FUNCTION_BLOCK FB_PressSectionDriveControl_V2_bak

VAR_INPUT

    //────────────────────────────────────────────
    // GROUP / INTERLOCKS
    //────────────────────────────────────────────
    startGroup              : BOOL; // Start command (pulse) / Comando de partida (pulso)
    stopGroup               : BOOL; // Stop command (level) / Comando de parada (nível)
    groupReset              : BOOL; // Fault reset / Reset de falhas do grupo
	
    //────────────────────────────────────────────
    // AUXILIARY MOTORS — INDICATORS & COMMANDS
    //────────────────────────────────────────────
    grouSpeedDifIncCmd         : BOOL; // Lamp: offset increasing / Lâmpada: aumento de offset
    grouSpeedDifDecCmd         : BOOL; // Lamp: offset decreasing / Lâmpada: redução de offset
	
    //────────────────────────────────────────────
    // SPEED ADJUSTMENTS / OFFSET TUNING
    //────────────────────────────────────────────
    groupRecoverSpeedCmd    : BOOL; // Recover speed while TRUE / Recuperar velocidade enquanto TRUE


    //────────────────────────────────────────────
    // DRIVE STATUS INPUTS — PRESS SECTION (2 MOTORS)
    //────────────────────────────────────────────
    firstPressReady         : BOOL; // First press (MASTER) ready / Prensa 1 (mestre) pronto
    secondPressReady        : BOOL; // Second press (SLAVE) ready / Prensa 2 (escravo) pronto

    //────────────────────────────────────────────
    // SPEED SETPOINTS / MODE
    //────────────────────────────────────────────
    groupAutoSpeedMPM       : REAL; // Auto mode speed [m/min] / Velocidade em modo automático [m/min]
    groupManualSpeedMPM     : REAL := 50.0; // Manual mode speed / Velocidade em modo manual
    groupSpeedAutoMan       : BOOL; // Speed mode: 0=Manual, 1=Auto / Modo de velocidade: 0=Manual, 1=Automático

    //────────────────────────────────────────────
    // SPEED & TORQUE FEEDBACKS
    //────────────────────────────────────────────
    firstPressSpeedFeedback : REAL; // First press speed feedback / Velocidade medida da prensa 1
    firstPressTorqueFeedback: REAL; // First press torque feedback / Torque da prensa 1
    secondPressSpeedFeedback: REAL; // Second press speed feedback / Velocidade medida da prensa 2
    secondPressTorqueFeedback: REAL; // Second press torque feedback / Torque da prensa 2


    //──── Upper Felt 1 Stretcher ────
    upperFelt1StretcherCmdFwd     : BOOL; // Run forward / Comando para frente
    upperFelt1StretcherCmdRev     : BOOL; // Run reverse / Comando para trás
    upperFelt1StretcherFault      : BOOL; // Fault detected / Falha detectada
    upperFelt1StretcherLimitFwd   : BOOL; // End limit forward / Fim de curso frente
    upperFelt1StretcherLimitRev   : BOOL; // End limit reverse / Fim de curso trás

    //──── Upper Felt 2 Stretcher ────
    upperFelt2StretcherCmdFwd     : BOOL; // Run forward / Comando para frente
    upperFeltt2tretcherCmdRev     : BOOL; // Run reverse / Comando para trás (corrigir nome!)
    upperFeltS2tretcherFault      : BOOL; // Fault detected / Falha detectada
    upperFeltS2tretcherLimitFwd   : BOOL; // End limit forward / Fim de curso frente
    upperFeltS2tretcherLimitRev   : BOOL; // End limit reverse / Fim de curso trás

    //──── Lower Felt Stretcher ────
    lowerFeltStretcherCmdFwd      : BOOL;
    lowerFeltStretcherCmdRev      : BOOL;
    lowerFeltStretcherFault       : BOOL;
    lowerFeltStretcherLimitFwd    : BOOL;
    lowerFeltStretcherLimitRev    : BOOL;

    //──── Upper Infeed Roll ────
    upperInfeedRollCmdFwd         : BOOL;
    upperInfeedRollCmdRev         : BOOL;
    upperInfeedRollFault          : BOOL;
    upperInfeedRollLimitFwd       : BOOL;
    upperInfeedRollLimitRev       : BOOL;

    //──── Lower Infeed Roll ────
    lowerInfeedRollCmdFwd         : BOOL;
    lowerInfeedRollCmdRev         : BOOL;
    lowerInfeedRollFault          : BOOL;
    lowerInfeedRollLimitFwd       : BOOL;
    lowerInfeedRollLimitRev       : BOOL;

    //────────────────────────────────────────────
    // FELT EDGE / RUNNING SAFETY SENSORS
    //────────────────────────────────────────────
    pressSectionUpperFelt1OverrunSensorOperatorSide : BOOL; // Operator side / Lado operador
    pressSectionUpperFelt1OverrunSensorDriveSide    : BOOL; // Drive side / Lado comando

    pressSectionUpperFelt2OverrunSensorOperatorSide : BOOL;
    pressSectionUpperFelt2OverrunSensorDriveSide    : BOOL;

    pressSectionLowerFeltOverrunSensorOperatorSide  : BOOL;
    pressSectionLowerFeltOverrunSensorDriveSide     : BOOL;

	
	machineConfig			:  PaperMachine_TypeHmiConfig;
	
END_VAR



VAR_OUTPUT

    //────────────────────────────────────────────
    // STATE / DIAGNOSTICS
    //────────────────────────────────────────────
    deviceState                 : STRING; // Current state string / Estado atual em texto
    statusCode                  : INT;    // 0=Idle, 1=Starting, 2=Running, 3=Fault
    groupFault                  : BOOL;   // TRUE if any group fault active / Falha geral do grupo


    //────────────────────────────────────────────
    // SPEED REFERENCES (TO DRIVES) AND DISPLAY
    //────────────────────────────────────────────
    firstPressSpeedSetpointRPM  		: REAL; // Master speed reference [%] / Referência de velocidade mestre
    secondPressSpeedSetpointRPM 		: REAL; // Slave speed reference [%] / Referência de velocidade escravo 
	
	firstPressSpeedFeedbackRPM  		: REAL; // Master speed reference [%] / Referência de velocidade mestre
    secondPressSpeedFeedbackRPM 		: REAL; // Slave speed reference [%] / Referência de velocidade escravo 
	
	firstPressSpeedFeedbackMPM  		: REAL; // Master speed reference [%] / Referência de velocidade mestre
    secondPressSpeedFeedbackMPM 		: REAL; // Slave speed reference [%] / Referência de velocidade escravo 

	firstPressTorqueFeedbackPct  		: REAL; // Master speed reference [%] / Referência de velocidade mestre
    secondPressTorqueFeedbackPct 		: REAL; // Slave speed reference [%] / Referência de velocidade escravo 
	
	
	nextGroupSpeedRefMPM        : REAL; // Next group speed [m/min] / Velocidade do próximo grupo [m/min]

    //────────────────────────────────────────────
    // TORQUE REFERENCES / LIMITS (SLAVE)
    //────────────────────────────────────────────
    firstPressTorqueRefPct : REAL; // Torque setpoint for slave / Referência de torque escravo

    //────────────────────────────────────────────
    // DRIVE COMMANDS (ENABLE / RESET)
    //────────────────────────────────────────────
    firstPressDriveEnable        : BOOL; // Enable master drive / Habilita drive mestre
    firstPressDriveReset         : BOOL; // Reset master drive fault / Reset falha drive mestre
    secondPressDriveEnable       : BOOL; // Enable slave drive / Habilita drive escravo
    secondPressDriveReset        : BOOL; // Reset slave drive fault / Reset falha drive escravo

    //────────────────────────────────────────────
    // STATUS CODES (PER DRIVE)
    //────────────────────────────────────────────
    firstPressStatusCode        : INT; // 0=Idle, 1=Start, 2=Run, 3=Fault / Código de status da prensa 1
    secondPressStatusCode       : INT; // Código de status da prensa 2

    //────────────────────────────────────────────
    // AUXILIARY MOTORS — DIRECT START OUTPUTS
    //────────────────────────────────────────────
    upperFelt1StretcherRunFwd   : BOOL; // Run forward / Rodar para frente
    upperFelt1StretcherRunRev   : BOOL; // Run reverse / Rodar para trás

    upperFelt2StretcherRunFwd   : BOOL;
    upperFelt2StretcherRunRev   : BOOL;

    lowerFeltStretcherRunFwd    : BOOL;
    lowerFeltStretcherRunRev    : BOOL;

    upperInfeedRollRunFwd       : BOOL;
    upperInfeedRollRunRev       : BOOL;

    lowerInfeedRollRunFwd       : BOOL;
    lowerInfeedRollRunRev       : BOOL;

    //────────────────────────────────────────────
    // HMI ALARMS STRUCTURE
    //────────────────────────────────────────────
    hmiAlarms                   : PaperMachine_TypeHmiAlarms; // Alarm structure / Estrutura de alarmes

END_VAR




VAR
 
	instFB_GroupDriveControl_V1 : FB_GroupDriveControl_V1;
	instFB_GroupSpeedControl_V1 : FB_GroupSpeedControl_V1;
	instFB_GroupDisplayFilters_V1 : FB_GroupDisplayFilters_V1;
	instFB_GroupTorqueTrimControl_V1 : FB_GroupTorqueTrimControl_V1;

	instFB_GroupTorqueTrimControl_V2: FB_GroupTorqueTrimControl_V2;
	speedDif: REAL;
	speedDifError: BOOL;
END_VAR

VAR PERSISTENT

END_VAR

// ─────────────────────────────────────────────────────────────────────────────
// MAIN CALL SEQUENCE
// ─────────────────────────────────────────────────────────────────────────────

_GroupControl();          // 1) State machine: edges, enables, stop modes
_StateDisplay();
_SpeedDifferenceCheck();  // 4) Speed difference monitor & trip
_auxiliaryControls();

_alarmsDisplay();

METHOD _alarmsDisplay
VAR_INPUT
END_VAR
(*
//==============================================================
// FAULT EVALUATION — PER CONDITION (flags only; no global set)
//==============================================================

//----------------------------
// PRESS SECTION DRIVES
//----------------------------
hmiAlarms.pressSectionFirstPressFaultAlarm  := firstPressVfdFaultFeedback;
hmiAlarms.pressSectionSecondPressFaultAlarm := secondPressVfdFaultFeedback;

//----------------------------
// PRESS SECTION AUXILIARIES
//----------------------------
hmiAlarms.pressSectionUpperFeltStretcherFaultAlarm := upperFelt1StretcherFault;
hmiAlarms.pressSectionLowerFeltStretcherFaultAlarm := lowerFeltStretcherFault;
hmiAlarms.pressSectionUpperInfeedRollFaultAlarm    := upperInfeedRollFault;
hmiAlarms.pressSectionLowerInfeedRollFaultAlarm    := lowerInfeedRollFault;


//==============================================================
// PRESS SECTION — FELT EDGE OVERRUN ALARMS (DIRECT SENSORS)
//==============================================================

hmiAlarms.pressSectionUpperFelt1OverrunOperatorSideAlarm := pressSectionUpperFelt1OverrunSensorOperatorSide;
hmiAlarms.pressSectionUpperFelt1OverrunDriveSideAlarm    := pressSectionUpperFelt1OverrunSensorDriveSide;

hmiAlarms.pressSectionUpperFelt2OverrunOperatorSideAlarm := pressSectionUpperFelt2OverrunSensorOperatorSide;
hmiAlarms.pressSectionUpperFelt2OverrunDriveSideAlarm    := pressSectionUpperFelt2OverrunSensorDriveSide;

hmiAlarms.pressSectionLowerFeltOverrunOperatorSideAlarm := pressSectionLowerFeltOverrunSensorOperatorSide;
hmiAlarms.pressSectionLowerFeltOverrunDriveSideAlarm    := pressSectionLowerFeltOverrunSensorDriveSide;


//----------------------------
// PRESS SECTION GROUP FAULT STATUS
//----------------------------
groupFault :=
    hmiAlarms.pressSectionFirstPressFaultAlarm 
	OR hmiAlarms.pressSectionSecondPressFaultAlarm 
	OR hmiAlarms.pressFelt1OverrunOperatorSideAlarm
	OR hmiAlarms.pressFelt1OverrunDriveSideAlarm
	OR hmiAlarms.pressFelt2OverrunOperatorSideAlarm
	OR hmiAlarms.pressFelt2OverrunDriveSideAlarm
	OR hmiAlarms.pressFelt3OverrunOperatorSideAlarm
	OR hmiAlarms.pressFelt3OverrunDriveSideAlarm;


*)
//==============================================================
// FAULT EVALUATION — PER CONDITION (flags only; no global set)
//==============================================================

//----------------------------
// PRESS SECTION DRIVES
//----------------------------
//hmiAlarms.pressSectionFirstPressFaultAlarm  := firstPressVfdFaultFeedback;
//hmiAlarms.pressSectionSecondPressFaultAlarm := secondPressVfdFaultFeedback;

//----------------------------
// PRESS SECTION AUXILIARIES
//----------------------------
hmiAlarms.pressSectionUpperFeltStretcherFaultAlarm := upperFelt1StretcherFault;
hmiAlarms.pressSectionLowerFeltStretcherFaultAlarm := lowerFeltStretcherFault;
hmiAlarms.pressSectionUpperInfeedRollFaultAlarm    := upperInfeedRollFault;
hmiAlarms.pressSectionLowerInfeedRollFaultAlarm    := lowerInfeedRollFault;


//==============================================================
// PRESS SECTION — FELT EDGE OVERRUN ALARMS (DIRECT SENSORS)
//==============================================================

hmiAlarms.pressSectionUpperFelt1OverrunOperatorSideAlarm := pressSectionUpperFelt1OverrunSensorOperatorSide;
hmiAlarms.pressSectionUpperFelt1OverrunDriveSideAlarm    := pressSectionUpperFelt1OverrunSensorDriveSide;

hmiAlarms.pressSectionUpperFelt2OverrunOperatorSideAlarm := pressSectionUpperFelt2OverrunSensorOperatorSide;
hmiAlarms.pressSectionUpperFelt2OverrunDriveSideAlarm    := pressSectionUpperFelt2OverrunSensorDriveSide;

hmiAlarms.pressSectionLowerFeltOverrunOperatorSideAlarm := pressSectionLowerFeltOverrunSensorOperatorSide;
hmiAlarms.pressSectionLowerFeltOverrunDriveSideAlarm    := pressSectionLowerFeltOverrunSensorDriveSide;


//----------------------------
// PRESS SECTION GROUP FAULT STATUS
//----------------------------
groupFault := hmiAlarms.pressSectionFirstPressFaultAlarm OR
		hmiAlarms.pressSectionSecondPressFaultAlarm OR
		hmiAlarms.pressSectionUpperFelt1OverrunOperatorSideAlarm OR
		hmiAlarms.pressSectionUpperFelt1OverrunDriveSideAlarm OR
		hmiAlarms.pressSectionUpperFelt2OverrunOperatorSideAlarm OR
		hmiAlarms.pressSectionUpperFelt2OverrunDriveSideAlarm OR
		hmiAlarms.pressSectionLowerFeltOverrunOperatorSideAlarm OR
		hmiAlarms.pressSectionLowerFeltOverrunDriveSideAlarm;
END_METHOD

METHOD _auxiliaryControls
VAR_INPUT
END_VAR
//============================
// LOWER FELT STRETCHER
//============================
IF NOT lowerFeltStretcherFault THEN
    IF lowerFeltStretcherCmdFwd AND NOT lowerFeltStretcherCmdRev AND NOT lowerFeltStretcherLimitFwd THEN
        lowerFeltStretcherRunFwd := TRUE;
    ELSE
        lowerFeltStretcherRunFwd := FALSE;
    END_IF;

    IF lowerFeltStretcherCmdRev AND NOT lowerFeltStretcherCmdFwd AND NOT lowerFeltStretcherLimitRev THEN
        lowerFeltStretcherRunRev := TRUE;
    ELSE
        lowerFeltStretcherRunRev := FALSE;
    END_IF;
ELSE
    lowerFeltStretcherRunFwd := FALSE;
    lowerFeltStretcherRunRev := FALSE;
END_IF;


//============================
// UPPER INFEED ROLL
//============================
IF NOT upperInfeedRollFault THEN
    IF upperInfeedRollCmdFwd AND NOT upperInfeedRollCmdRev AND NOT upperInfeedRollLimitFwd THEN
        upperInfeedRollRunFwd := TRUE;
    ELSE
        upperInfeedRollRunFwd := FALSE;
    END_IF;

    IF upperInfeedRollCmdRev AND NOT upperInfeedRollCmdFwd AND NOT upperInfeedRollLimitRev THEN
        upperInfeedRollRunRev := TRUE;
    ELSE
        upperInfeedRollRunRev := FALSE;
    END_IF;
ELSE
    upperInfeedRollRunFwd := FALSE;
    upperInfeedRollRunRev := FALSE;
END_IF;


//============================
// LOWER INFEED ROLL
//============================
IF NOT lowerInfeedRollFault THEN
    IF lowerInfeedRollCmdFwd AND NOT lowerInfeedRollCmdRev AND NOT lowerInfeedRollLimitFwd THEN
        lowerInfeedRollRunFwd := TRUE;
    ELSE
        lowerInfeedRollRunFwd := FALSE;
    END_IF;

    IF lowerInfeedRollCmdRev AND NOT lowerInfeedRollCmdFwd AND NOT lowerInfeedRollLimitRev THEN
        lowerInfeedRollRunRev := TRUE;
    ELSE
        lowerInfeedRollRunRev := FALSE;
    END_IF;
ELSE
    lowerInfeedRollRunFwd := FALSE;
    lowerInfeedRollRunRev := FALSE;
END_IF;


//============================
// UPPER FELT 1 STRETCHER
//============================
IF NOT upperFelt1StretcherFault THEN
    IF upperFelt1StretcherCmdFwd AND NOT upperFelt1StretcherCmdRev AND NOT upperFelt1StretcherLimitFwd THEN
        upperFelt1StretcherRunFwd := TRUE;
    ELSE
        upperFelt1StretcherRunFwd := FALSE;
    END_IF;

    IF upperFelt1StretcherCmdRev AND NOT upperFelt1StretcherCmdFwd AND NOT upperFelt1StretcherLimitRev THEN
        upperFelt1StretcherRunRev := TRUE;
    ELSE
        upperFelt1StretcherRunRev := FALSE;
    END_IF;
ELSE
    upperFelt1StretcherRunFwd := FALSE;
    upperFelt1StretcherRunRev := FALSE;
END_IF;

//============================
// UPPER FELT 2 STRETCHER
//============================
IF NOT upperFeltS2tretcherFault THEN
    IF upperFelt2StretcherCmdFwd AND NOT upperFeltt2tretcherCmdRev AND NOT upperFeltS2tretcherLimitFwd THEN
        upperFelt2StretcherRunFwd := TRUE;
    ELSE
        upperFelt2StretcherRunFwd := FALSE;
    END_IF;

    IF upperFeltt2tretcherCmdRev AND NOT upperFelt2StretcherCmdFwd AND NOT upperFeltS2tretcherLimitRev THEN
        upperFelt2StretcherRunRev := TRUE;
    ELSE
        upperFelt2StretcherRunRev := FALSE;
    END_IF;
ELSE
    upperFelt2StretcherRunFwd := FALSE;
    upperFelt2StretcherRunRev := FALSE;
END_IF;
END_METHOD

METHOD _GroupControl
VAR_INPUT
END_VAR
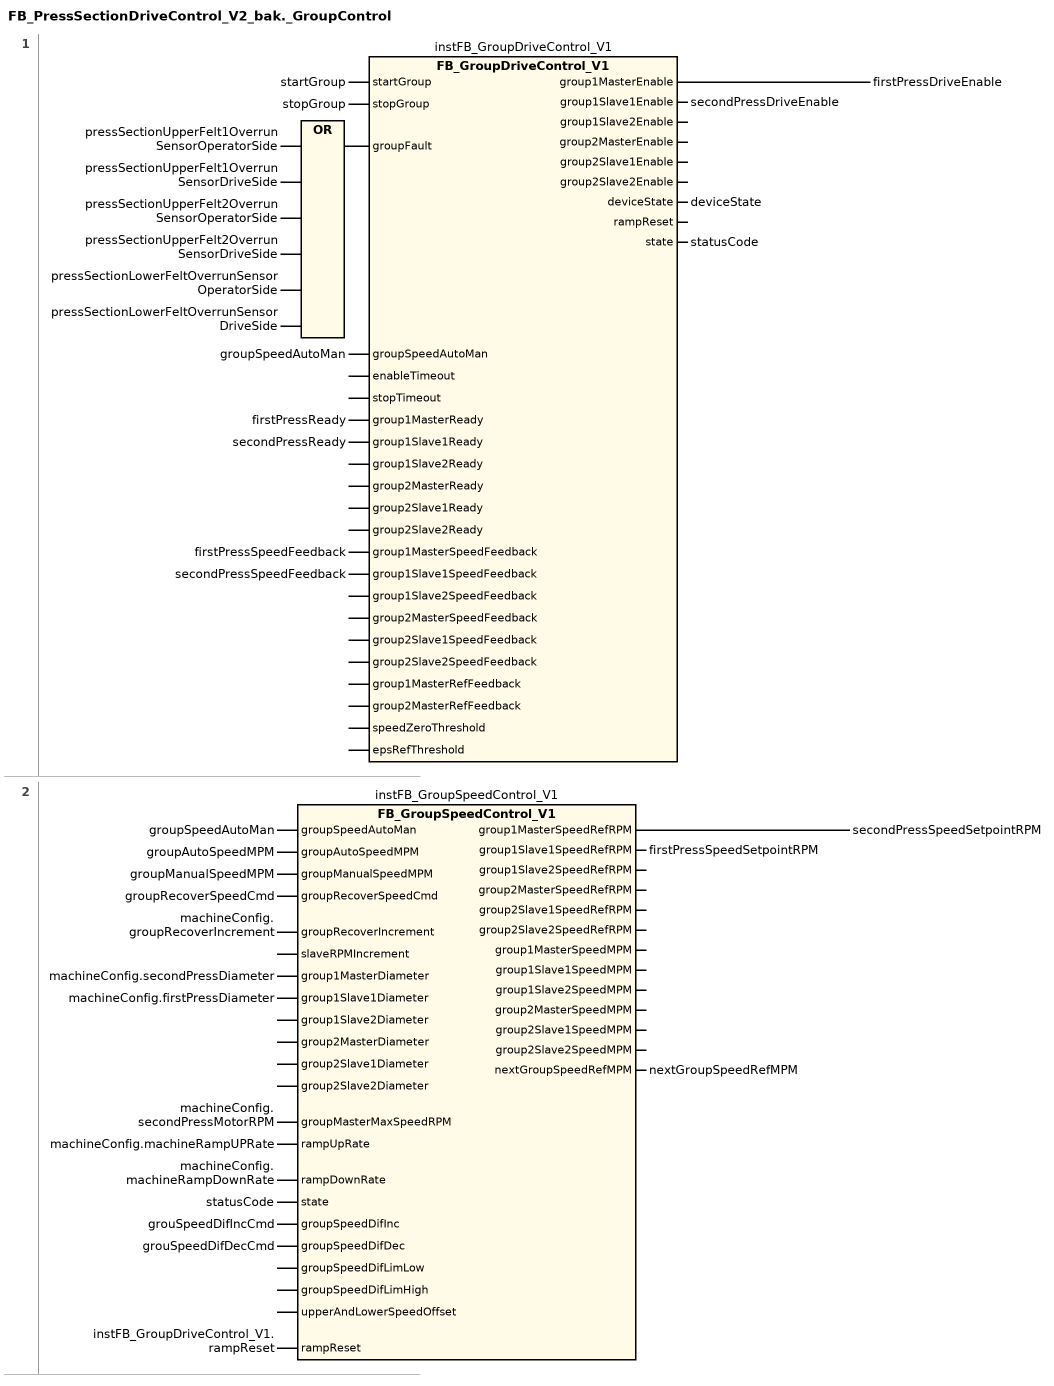
// NETWORK 1
instFB_GroupDriveControl_V1(
    startGroup := startGroup,
    stopGroup := stopGroup,
    groupFault := pressSectionUpperFelt1OverrunSensorOperatorSide OR pressSectionUpperFelt1OverrunSensorDriveSide OR pressSectionUpperFelt2OverrunSensorOperatorSide OR pressSectionUpperFelt2OverrunSensorDriveSide OR pressSectionLowerFeltOverrunSensorOperatorSide OR pressSectionLowerFeltOverrunSensorDriveSide,
    groupSpeedAutoMan := groupSpeedAutoMan,
    group1MasterReady := firstPressReady,
    group1Slave1Ready := secondPressReady,
    group1MasterSpeedFeedback := firstPressSpeedFeedback,
    group1Slave1SpeedFeedback := secondPressSpeedFeedback,
    group1Slave1Enable => secondPressDriveEnable,
    deviceState => deviceState,
    state => statusCode); // FB_GroupDriveControl_V1
firstPressDriveEnable := instFB_GroupDriveControl_V1.group1MasterEnable;

// NETWORK 2
instFB_GroupSpeedControl_V1(
    groupSpeedAutoMan := groupSpeedAutoMan,
    groupAutoSpeedMPM := groupAutoSpeedMPM,
    groupManualSpeedMPM := groupManualSpeedMPM,
    groupRecoverSpeedCmd := groupRecoverSpeedCmd,
    groupRecoverIncrement := machineConfig.groupRecoverIncrement,
    group1MasterDiameter := machineConfig.secondPressDiameter,
    group1Slave1Diameter := machineConfig.firstPressDiameter,
    groupMasterMaxSpeedRPM := machineConfig.secondPressMotorRPM,
    rampUpRate := machineConfig.machineRampUPRate,
    rampDownRate := machineConfig.machineRampDownRate,
    state := statusCode,
    groupSpeedDifInc := grouSpeedDifIncCmd,
    groupSpeedDifDec := grouSpeedDifDecCmd,
    rampReset := instFB_GroupDriveControl_V1.rampReset,
    group1Slave1SpeedRefRPM => firstPressSpeedSetpointRPM,
    nextGroupSpeedRefMPM => nextGroupSpeedRefMPM); // FB_GroupSpeedControl_V1
secondPressSpeedSetpointRPM := instFB_GroupSpeedControl_V1.group1MasterSpeedRefRPM;

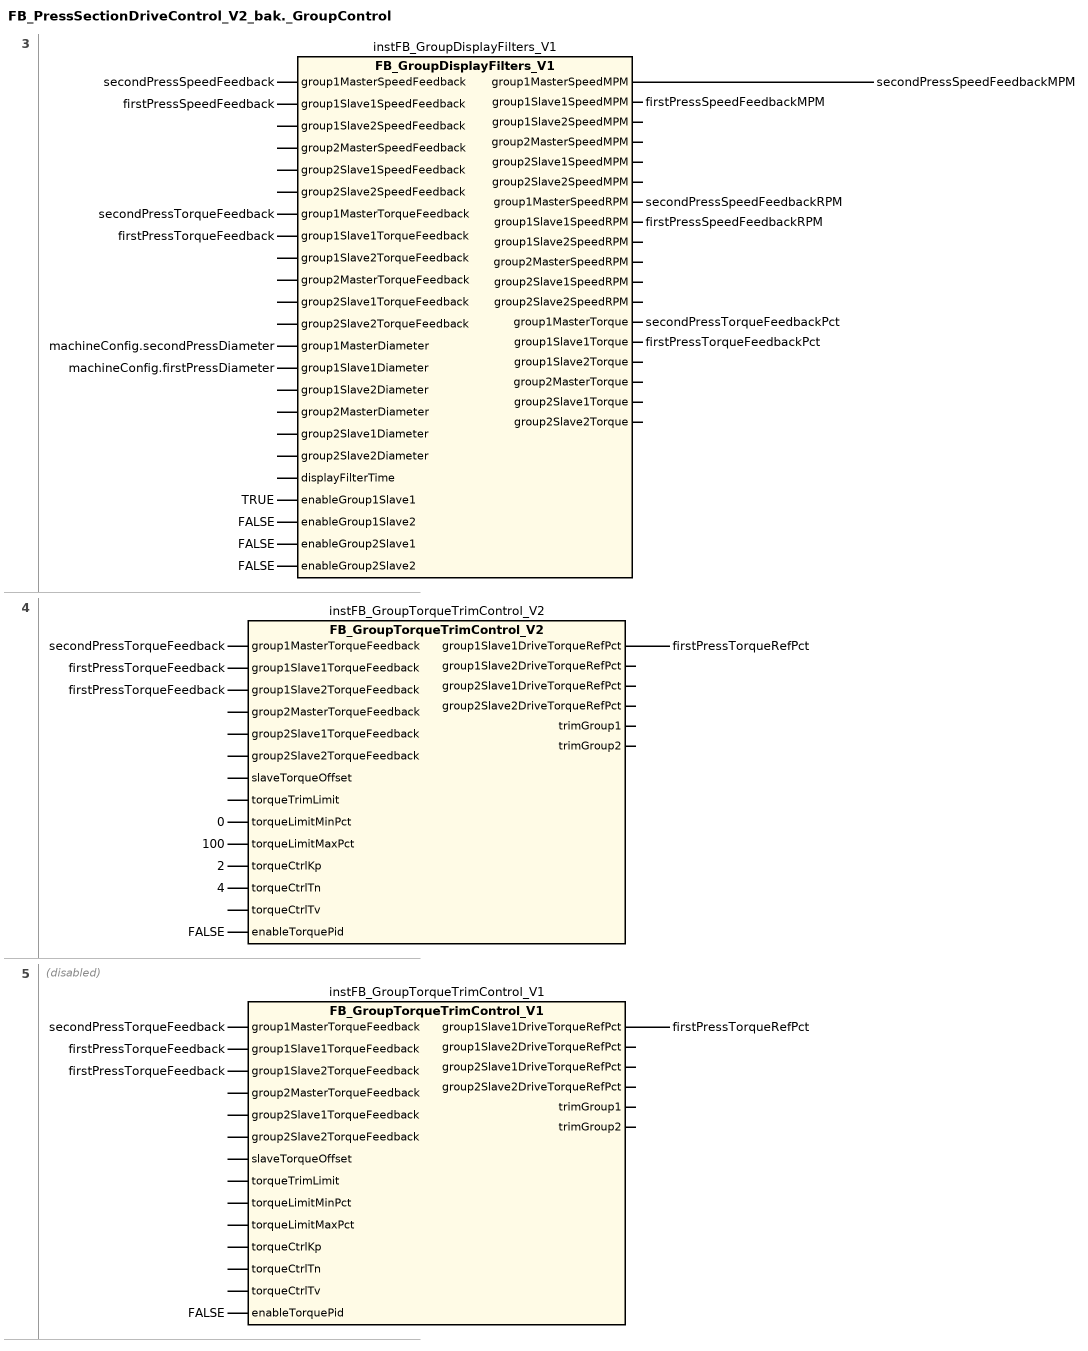
// NETWORK 3
instFB_GroupDisplayFilters_V1(
    group1MasterSpeedFeedback := secondPressSpeedFeedback,
    group1Slave1SpeedFeedback := firstPressSpeedFeedback,
    group1MasterTorqueFeedback := secondPressTorqueFeedback,
    group1Slave1TorqueFeedback := firstPressTorqueFeedback,
    group1MasterDiameter := machineConfig.secondPressDiameter,
    group1Slave1Diameter := machineConfig.firstPressDiameter,
    enableGroup1Slave1 := TRUE,
    enableGroup1Slave2 := FALSE,
    enableGroup2Slave1 := FALSE,
    enableGroup2Slave2 := FALSE,
    group1Slave1SpeedMPM => firstPressSpeedFeedbackMPM,
    group1MasterSpeedRPM => secondPressSpeedFeedbackRPM,
    group1Slave1SpeedRPM => firstPressSpeedFeedbackRPM,
    group1MasterTorque => secondPressTorqueFeedbackPct,
    group1Slave1Torque => firstPressTorqueFeedbackPct); // FB_GroupDisplayFilters_V1
secondPressSpeedFeedbackMPM := instFB_GroupDisplayFilters_V1.group1MasterSpeedMPM;

// NETWORK 4
instFB_GroupTorqueTrimControl_V2(
    group1MasterTorqueFeedback := secondPressTorqueFeedback,
    group1Slave1TorqueFeedback := firstPressTorqueFeedback,
    group1Slave2TorqueFeedback := firstPressTorqueFeedback,
    torqueLimitMinPct := 0,
    torqueLimitMaxPct := 100,
    torqueCtrlKp := 2,
    torqueCtrlTn := 4,
    enableTorquePid := FALSE); // FB_GroupTorqueTrimControl_V2
firstPressTorqueRefPct := instFB_GroupTorqueTrimControl_V2.group1Slave1DriveTorqueRefPct;

// NETWORK 5 (disabled)
// instFB_GroupTorqueTrimControl_V1(
//     group1MasterTorqueFeedback := secondPressTorqueFeedback,
//     group1Slave1TorqueFeedback := firstPressTorqueFeedback,
//     group1Slave2TorqueFeedback := firstPressTorqueFeedback,
//     enableTorquePid := FALSE); // FB_GroupTorqueTrimControl_V1
// firstPressTorqueRefPct := instFB_GroupTorqueTrimControl_V1.group1Slave1DriveTorqueRefPct;
END_METHOD

METHOD PRIVATE _Scale : REAL
VAR_INPUT
    X    : REAL;
    I_LO : REAL;
    I_HI : REAL;
    O_LO : REAL;
    O_HI : REAL;
END_VAR
IF I_LO = I_HI THEN
	_Scale := O_LO;
ELSE
	_Scale := (O_HI - O_LO) / (I_HI - I_LO) * (LIMIT(I_LO, X, I_HI) - I_LO) + O_LO;
END_IF;
END_METHOD

// ============================== Methods ==============================
// Intra-section speed supervision for Press Section (firstPress ↔ secondPress)
METHOD _SpeedDifferenceCheck
VAR_INPUT
END_VAR
VAR
    diffPress : REAL;   // Absolute speed difference between master and slave
END_VAR

(*
    //────────────────────────────────────────────
    firstPressSpeedFeedback : REAL; // First press speed feedback / Velocidade medida da prensa 1
    firstPressTorqueFeedback: REAL; // First press torque feedback / Torque da prensa 1
    secondPressSpeedFeedback: REAL; // Second press speed feedback / Velocidade medida da prensa 2
    secondPressTorqueFeedback: REAL; // Second press torque feedback / Torque da prensa 2

*)


speedDif := ABS(firstPressSpeedFeedback - secondPressSpeedFeedback);


IF speedDif > 10 THEN
	
	speedDifError := TRUE;
	
	ELSE
		
	speedDifError := FALSE;
	
	
END_IF
END_METHOD

METHOD _StateDisplay
VAR_INPUT
END_VAR

// ──────────────────────────────────────────────────────────────────────────────
// _StateDisplay — Press Section (firstPress = Master, secondPress = Slave)
// Maps the internal machine "state" to a compact HMI status code and derives
// per-drive motor status codes from VFD signals.
//
// statusCode / firstPressStatusCode / secondPressStatusCode legend:
//   0 = Idle, 1 = Starting, 2 = Running, 3 = Fault
//
// Machine "state" groups:
//   0 = IDLE, 1 = ENABLE, 2 = WAIT_EN, 3 = RAMP_EN, 4 = RUN, 5 = STOPPING, 10 = FAULT
// Priority rule (for motors): Fault > Running > Starting > Idle
// ──────────────────────────────────────────────────────────────────────────────
VAR CONSTANT
    STATUS_IDLE     : INT := 0;
    STATUS_STARTING : INT := 1;
    STATUS_RUNNING  : INT := 2;
    STATUS_FAULT    : INT := 3;
END_VAR
(*
// ─────────────── Group machine states into a single HMI statusCode ───────────
CASE state OF
    10: // FAULT
        statusCode := STATUS_FAULT;
    4:  // RUN
        statusCode := STATUS_RUNNING;
    1, 2, 3: // ENABLE / WAIT_EN / RAMP_EN
        statusCode := STATUS_STARTING;
ELSE   // IDLE, STOPPING, or any other
        statusCode := STATUS_IDLE;
END_CASE;


// ─────────────── Per-drive status (priority: Fault > Running > Starting > Idle) ───────────────
// FIRST PRESS (MASTER)
IF firstPressVfdFaultFeedback THEN
    firstPressStatusCode := STATUS_FAULT;
ELSIF firstPressVfdRunFeedback THEN
    firstPressStatusCode := STATUS_RUNNING;
ELSIF firstPressDriveEnable THEN
    firstPressStatusCode := STATUS_STARTING;
ELSE
    firstPressStatusCode := STATUS_IDLE;
END_IF;

// SECOND PRESS (SLAVE)
IF secondPressVfdFaultFeedback THEN
    secondPressStatusCode := STATUS_FAULT;
ELSIF secondPressVfdRunFeedback THEN
    secondPressStatusCode := STATUS_RUNNING;
ELSIF secondPressDriveEnable THEN
    secondPressStatusCode := STATUS_STARTING;
ELSE
    secondPressStatusCode := STATUS_IDLE;
END_IF;
*)
END_METHOD

END_FUNCTION_BLOCK

(* stored: Version 1.1.0.1, ProductVersion 3.1.4024.15
   POU FB_PressSectionDriveControl_V2_bak: Id {b4fc8681-3b45-4b8f-a60d-b34f273b6ce7}, SpecialFunc None
   Method _alarmsDisplay: Id {b0deda9d-f19c-4cf5-b28d-2e913bc34b83}
   Method _auxiliaryControls: Id {dd958152-4880-4c0a-acb2-95912180848d}
   Method _GroupControl: Id {a30edc36-99d4-48b4-8d2d-308480737910}
   Method _Scale: Id {4f1b9d3a-1608-4b84-b643-27a0c97068aa}
   Method _SpeedDifferenceCheck: Id {8c1e15bc-a81c-48ce-9ab6-034745ca4061}
   Method _StateDisplay: Id {7600a825-fdf6-4759-954f-a30b8aaeea1a} *)
